// TIA Portal V18 export
FUNCTION_BLOCK "BLINKER"   // FB30, LAD
{ S7_Optimized_Access := 'TRUE' }
VERSION : 0.1
// stored: AutoNumber true, IsIECCheckEnabled false, IsRetainMemResEnabled false, MemoryReserve 100, SetENOAutomatically false, UDAEnableTagReadback false
   VAR_INPUT
      BLINK_NOW : Bool;
      ON_t : Time := T#10s;
      OFF_t : Time := T#10s;
   END_VAR
   VAR_OUTPUT
      yToBlink : Bool;
   END_VAR
   VAR
      tON_DB { S7_SetPoint := 'True'} : TON_TIME;
      tOFF_DB { S7_SetPoint := 'True'} : TON_TIME;
      off_mem { S7_SetPoint := 'True'} : Bool;
   END_VAR
   VAR_TEMP   // added for the SCL form of the ladder/FBD networks
      _w1 : Bool;
   END_VAR
BEGIN

REGION Network 1
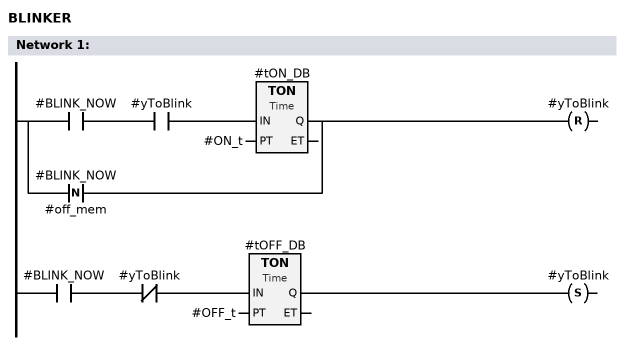
   RUNG wire#powerrail
      Contact( #BLINK_NOW )
      Contact( #yToBlink )
      { S7_Templates := "time_type := Time" } #tON_DB.TON(pt := #ON_t, et =>)
      wire#w1
      R_Coil( #yToBlink )
   END_RUNG
   RUNG wire#powerrail
      N_Contact(operand := #BLINK_NOW, bit := #off_mem)
   END_RUNG wire#w1
   RUNG wire#powerrail
      Contact( #BLINK_NOW )
      I_Contact( #yToBlink )
      { S7_Templates := "time_type := Time" } #tOFF_DB.TON(pt := #OFF_t, et =>)
      S_Coil( #yToBlink )
   END_RUNG
   // the same network as SCL:
   #tON_DB(IN := #BLINK_NOW AND #yToBlink, PT := #ON_t);   // TON
   #_w1 := NOT #BLINK_NOW AND #off_mem;   // falling edge of #BLINK_NOW
   #off_mem := #BLINK_NOW;
   IF #tON_DB.Q OR #_w1 THEN #yToBlink := FALSE; END_IF;
   #tOFF_DB(IN := #BLINK_NOW AND NOT #yToBlink, PT := #OFF_t);   // TON
   IF #tOFF_DB.Q THEN #yToBlink := TRUE; END_IF;
END_REGION
END_FUNCTION_BLOCK
